// TIA Portal V15.1 export
// export: Created 2022-11-23T22:00:00.6184614Z, ExportSetting WithDefaults, WithReadOnly, DisplayName Totally Integrated Automation Portal, DisplayVersion V15.1 Update 5, DisplayName TIA Portal Openness, DisplayVersion V15.1 Update 5, DisplayName STEP 7 Professional, DisplayVersion V15.1 Update 5, DisplayName WinCC Advanced, DisplayVersion V15.1 Update 5
FUNCTION_BLOCK "Automacao_de_teste"   // FB1, LAD
{ S7_Optimized_Access := 'TRUE' }
VERSION : 0.1
// stored: AutoNumber true, CodeModifiedDate 2022-11-23T21:57:36.2825254Z, CompileDate 2022-11-23T21:57:38.1368966Z, CreationDate 2022-11-23T21:49:22.7073363Z, DownloadWithoutReinit false, HandleErrorsWithinBlock false, InterfaceModifiedDate 2022-11-23T21:54:21.9909482Z, IsConsistent true, IsIECCheckEnabled false, IsKnowHowProtected false, ISMultiInstanceCapable true, IsRetainMemResEnabled false, IsWriteProtected false, LibraryConformanceStatus The object is library-conformant., MemoryReserve 100, ModifiedDate 2022-11-23T21:57:36.2825254Z, ParameterModified 2022-11-23T21:54:21.9909482Z, PLCSimAdvancedSupport false, SetENOAutomatically False, StructureModified 2022-11-23T21:54:21.9909482Z, UDAEnableTagReadback false
   VAR_INPUT
      Tag1 : Bool;
      Tag2 : Bool;
      Tag3 : Bool;
      Tag4 : Bool;
      Tag10 : Bool;
      Tag11 : Bool;
      Tag12 : Bool;
      Tag13 : Bool;
      Tag14 : Bool;
   END_VAR
   VAR_OUTPUT
      Tag20 : Bool;
      Tag21 : Bool;
      Tag22 : Bool;
      Tag23 : Bool;
      Tag24 : Bool;
   END_VAR
   VAR_IN_OUT
      Tag5 : Bool;
      Tag6 : Bool;
      Tag7 : Bool;
      Tag8 : Bool;
      Tag9 : Bool;
   END_VAR
   VAR_TEMP   // added for the SCL form of the ladder/FBD networks
      _w1 : Bool;
   END_VAR
BEGIN

REGION Network 1
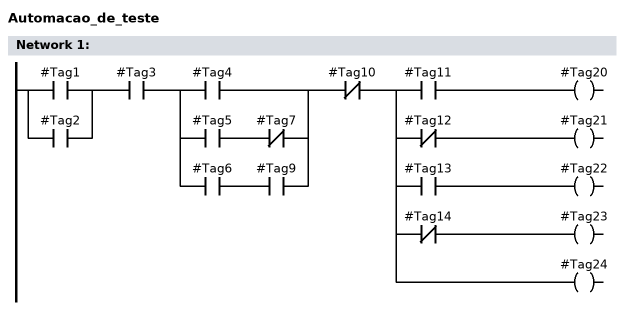
   RUNG wire#powerrail
      Contact( #Tag1 )
      wire#w1
      Contact( #Tag3 )
      wire#w2
      Contact( #Tag4 )
      wire#w3
      I_Contact( #Tag10 )
      wire#w4
      Contact( #Tag11 )
      Coil( #Tag20 )
   END_RUNG
   RUNG wire#powerrail
      Contact( #Tag2 )
   END_RUNG wire#w1
   RUNG wire#w2
      Contact( #Tag5 )
      I_Contact( #Tag7 )
   END_RUNG wire#w3
   RUNG wire#w2
      Contact( #Tag6 )
      Contact( #Tag9 )
   END_RUNG wire#w3
   RUNG wire#w4
      I_Contact( #Tag12 )
      Coil( #Tag21 )
   END_RUNG
   RUNG wire#w4
      Contact( #Tag13 )
      Coil( #Tag22 )
   END_RUNG
   RUNG wire#w4
      I_Contact( #Tag14 )
      Coil( #Tag23 )
   END_RUNG
   RUNG wire#w4
      Coil( #Tag24 )
   END_RUNG
   // the same network as SCL:
   #_w1 := (#Tag1 OR #Tag2) AND #Tag3 AND (#Tag4 OR (#Tag5 AND NOT #Tag7) OR (#Tag6 AND #Tag9)) AND NOT #Tag10;
   #Tag20 := #_w1 AND #Tag11;
   #Tag21 := #_w1 AND NOT #Tag12;
   #Tag22 := #_w1 AND #Tag13;
   #Tag23 := #_w1 AND NOT #Tag14;
   #Tag24 := #_w1;
END_REGION
END_FUNCTION_BLOCK
